// This function has been automatically generated from the project information.
{attribute 'signature_flag' := '1073741824'}
{attribute 'TcGenerated'}
{attribute 'no-analysis'}
FUNCTION F_GetTitle : WSTRING
VAR_INPUT
	
END_VAR

F_GetTitle := "Xts Library";

END_FUNCTION

(* stored: Version 1.1.0.1
   POU F_GetTitle: Id {ad995e86-7062-4cf6-b990-b2fc88f0d330}, SpecialFunc None *)
